(* CODESYS project MyCustomLib.library
   Company: MyCompany DERO
   DefaultNamespace: MyCustomLin
   Version: 0.1.0.0
   Placeholder: Custom
   Author: DejanRozic
   Description: Libary for FC and FB
   Title: Custom

Project tree, tasks and I/O mapping:
  libraries: Tc2_Standard, * (Beckhoff Automation GmbH); Tc2_System, * (Beckhoff Automation GmbH); Tc3_Module, * (Beckhoff Automation GmbH)
  DUTs/
    data type E_EventType
    data type ST_Event
    data type ST_HMI_CounterGlobalSettings
    data type ST_HMI_CounterGlobalSettings_1
    data type st_HMI_DigitalInputsDataGrid
    data type st_HMI_DigitalInputsDataGrid_1
    data type ST_HMI_GlobalCounter_Counters
    data type ST_HMI_GlobalCounter_Counters_1
  GVLs/
    POUs/
      COUNTERS/
        function block FB_GlobalCounter [ST]: M_ResetCounterToZero, P_isCounterFull
      TIME/
        function FC_GetLocalTime [ST]
      TIME_CONVERTION/
        function FC_UpdateEventTimeWIthSystemTime [ST]
      program MAIN [ST]
  Version/
    global variables Global_Version
  VISUs/
*)

// DUTs/E_EventType
{attribute 'qualified_only'}
{attribute 'strict'}
{attribute 'to_string'} //Atribbute to convert from enum to string!
TYPE E_EventType :
(
	Alarm := 0,
	Message
);
END_TYPE

// DUTs/ST_Event
TYPE ST_Event :
STRUCT
	eEventType		: E_EventType;
	eEventServerity	: TcEventSeverity;
	nEventIdenity	: UDINT;
	sEventText		: STRING(255); //mesage
	dtTimeStamp		: DATE_AND_TIME;
END_STRUCT
END_TYPE

// DUTs/ST_HMI_CounterGlobalSettings
TYPE ST_HMI_CounterGlobalSettings :
STRUCT
	uStKosovNaObrat :	UINT;
	uStObratovNaKos	:	UINT;
END_STRUCT
END_TYPE

// DUTs/ST_HMI_CounterGlobalSettings_1
TYPE ST_HMI_CounterGlobalSettings_1 :
STRUCT
	uStKosovNaObrat :	UINT;
	uStObratovNaKos	:	UINT;
END_STRUCT
END_TYPE

// DUTs/st_HMI_DigitalInputsDataGrid
TYPE st_HMI_DigitalInputsDataGrid :
STRUCT
	sCustomNameOfInput:		STRING; //Custom name of input
	xCurentInputStatus:		BOOL;	//Current Status of input 0-OFF, 1-ON
	xInputEnable:			BOOL;	//Input enable 0 - disable, 1 - enable
	iSensorType:			INT;	//Sensor Type 0-NO, 1-NC
	uAngleStart:			UINT;   //CAM Start Angle
	uAngleStop:				UINT;	//CAM Stop angle
	
END_STRUCT
END_TYPE

// DUTs/st_HMI_DigitalInputsDataGrid_1
TYPE st_HMI_DigitalOutputsDataGrid :
STRUCT
	sCusomNameOfInput:		STRING; //Custom name of input
	xCurentInputStatus:		BOOL;	//Current Status of input 0-OFF, 1-ON
	xInputEnable:			BOOL;	//Input enable 0 - disable, 1 - enable
	iSensorType:			INT;	//Sensor Type 0-NO, 1-NC
	uAngleStart:			UINT;   //CAM Start Angle
	uAngleStop:				UINT;	//CAM Stop angle
	uDynTime:				TIME;	//Time for dynamic output
	uKorak:					UINT;	// number of steps for actiavation
	
END_STRUCT
END_TYPE

// DUTs/ST_HMI_GlobalCounter_Counters
TYPE ST_HMI_GlobalCounter_Counters :
STRUCT
	stName					:   STRING;
	udCounterIzdelano		:   UDINT;
	udCounterZeljeno		:   UDINT;
	xCounterisEnabled		:	BOOL;
	xResetButtonIsPressed	:	BOOL;
	xCounterIsFULL			:	BOOL;
END_STRUCT
END_TYPE

// DUTs/ST_HMI_GlobalCounter_Counters_1
TYPE ST_HMI_GlobalCounter_Counters_1 :
STRUCT
	stName					:   STRING;
	udCounterIzdelano		:   UDINT;
	udCounterZeljeno		:   UDINT;
	xCounterisEnabled		:	BOOL;
	xResetButtonIsPressed	:	BOOL;
	xCounterIsFULL			:	BOOL;
END_STRUCT
END_TYPE

// Version/Global_Version
{attribute 'TcGenerated'}
{attribute 'no-analysis'}
{attribute 'linkalways'}
// This function has been automatically generated from the project information.
VAR_GLOBAL CONSTANT
	{attribute 'const_non_replaced'}
	stLibVersion_Custom : ST_LibVersion := (iMajor := 0, iMinor := 1, iBuild := 0, iRevision := 0, nFlags := 0, sVersion := '0.1.0.0');
END_VAR

// GVLs/POUs/COUNTERS/FB_GlobalCounter
FUNCTION_BLOCK FB_GlobalCounter
VAR_INPUT
	xTrigg 				:	BOOL;
	stGlobalCounter 	: REFERENCE TO ST_HMI_GlobalCounter_Counters;
	stCounterSettings 	: REFERENCE TO ST_HMI_CounterGlobalSettings;
END_VAR
VAR_OUTPUT
	xError : BOOL;
	xCounterIsFULL: BOOL;
END_VAR
VAR
	rtrig : ARRAY[0..5] OF R_TRIG;
	_CounterIsFULL : BOOL;
	_uCounterValue	:	 UINT;
	
END_VAR

//Nastvitev za robni pogoj
rtrig[0](CLK:=xTrigg);
rtrig[1](CLK:=stGlobalCounter.xResetButtonIsPressed);

//ce je counter <> 1 potem glej interni counter <--||-- 
//****************************************************
// 1. PREVERI če je  stObratovnaKos > 1
// 2. Če je večje prištej 1 internemu counterju in primerjaj z podano vrednostno
// 3. če ni večji samo prištej kose

IF stCounterSettings.uStObratovNaKos> 1 THEN
	IF rtrig[0].Q AND stGlobalCounter.xCounterisEnabled THEN
		_uCounterValue := _uCounterValue + 1; //pristej ena lokalnemo counterju		
		IF _uCounterValue >= stCounterSettings.uStObratovNaKos THEN // ce je counter >= kos/obrat potem pristej 1
			stGlobalCounter.udCounterIzdelano := stGlobalCounter.udCounterIzdelano + stCounterSettings.uStKosovNaObrat;
			_uCounterValue := 0; //reset lokalnega counterja
		END_IF
	END_IF 
ELSE
	IF rtrig[0].Q AND stGlobalCounter.xCounterisEnabled THEN 
	stGlobalCounter.udCounterIzdelano := stGlobalCounter.udCounterIzdelano + stCounterSettings.uStKosovNaObrat;  
	END_IF
END_IF


//reset števca
IF rtrig[1].Q THEN // RESET STEVCA
	M_ResetCounterToZero();
END_IF

//Javljanje napake - counter je FULL
IF stGlobalCounter.udCounterIzdelano >= stGlobalCounter.udCounterZeljeno THEN
	P_isCounterFull := TRUE;
ELSE
	P_isCounterFull := FALSE;
END_IF


//POSTAVITEV IZHODOV 
xCounterIsFULL := _CounterIsFULL;
xError := _CounterIsFULL;


//ZAPIS STRUKTURE - vpis da je counter FULL
stGlobalCounter.xCounterIsFULL := _CounterIsFULL;

METHOD M_ResetCounterToZero : BOOL
VAR_INPUT
END_VAR
stGlobalCounter.udCounterIzdelano := 0;
END_METHOD

PROPERTY PRIVATE P_isCounterFull : BOOL
GET
P_isCounterFull :=_CounterIsFULL;
END_GET
SET
_CounterIsFULL := P_isCounterFull;
END_SET
END_PROPERTY

END_FUNCTION_BLOCK

// GVLs/POUs/TIME/FC_GetLocalTime
FUNCTION FC_GetLocalTime : BOOL
VAR_INPUT
	sNetID	:	T_AmsNetID ;
    bEnable   : BOOL;
    dwCycle   : DWORD(1..86400) := 5;
    dwOpt     : DWORD := 1;
    tTimeout  : TIME := DEFAULT_ADS_TIMEOUT;
END_VAR
VAR
	fbGetLocalTime					:	FB_LocalSystemTime;	
	bValid							:	BOOL;
	tzID							:	E_TimeZoneID;
	
END_VAR
VAR_OUTPUT
	systemTime						:	TIMESTRUCT;
END_VAR

fbGetLocalTime(sNetID :=sNetID,
				bEnable := bEnable,
				dwCycle := dwCycle,
				tTimeout := tTimeout,
				bValid => bValid,
				tzID => tzID,				
				systemTime => systemTime);

END_FUNCTION

// GVLs/POUs/TIME_CONVERTION/FC_UpdateEventTimeWIthSystemTime
FUNCTION FC_UpdateEventTimeWIthSystemTime
VAR_INPUT
	stEvent : REFERENCE TO ST_Event;
END_VAR
VAR
	fbGetSystemTime	:	GETSYSTEMTIME; //SYSTEM TIME
	stFileTime : T_FILETIME;		//SAVE IT TO DT
END_VAR

fbGetSystemTime(timeHiDW=>stFileTime.dwHighDateTime, 
				timeLoDW =>stFileTime.dwLowDateTime); // Convert to DT
			
stEvent.dtTimeStamp:=FILETIME_TO_DT(fileTime:=stFileTime);

END_FUNCTION

// GVLs/POUs/MAIN
PROGRAM MAIN
VAR
END_VAR

END_PROGRAM
